PROGRAM MAIN
VAR
END_VAR

END_PROGRAM

(* stored: Version 1.1.0.1
   POU MAIN: Id {29649493-4e4b-4bdf-a4e4-7515b23769d2} *)
